{attribute 'qualified_only'}
VAR_GLOBAL CONSTANT
	DEFAULT_IPV4_ADDRESS	: Tc2_System.T_IPv4Addr := ;	// The default Ip address
	DEFAULT_PORT			: ZigaLibs_TcpIp.T_Port := 6363;	// The default port setting
END_VAR

(* stored: Version 1.1.0.1, ProductVersion 3.1.4024.15
   GVL GVL_EnduranceInfraredPyrometer: Id {41359764-71fc-073d-3481-d19f5d745722} *)
